INTERFACE I_Motor

METHOD Start : BOOL
VAR_INPUT
	force : BOOL;
END_VAR
END_METHOD

PROPERTY PUBLIC Speed : INT
GET
END_GET
END_PROPERTY

END_INTERFACE

(* stored: Version 1.1.0.1, ProductVersion 3.1.4026.18
   Itf I_Motor: Id {00000000-0000-0000-0000-000000000060}
   Method Start: Id {00000000-0000-0000-0000-000000000061}
   Property Speed: Id {00000000-0000-0000-0000-000000000062}
   Get Get: Id {00000000-0000-0000-0000-000000000063} *)
